FUNCTION_BLOCK CC1SFC
VAR_INPUT
	mode : UINT := 0; //0 = manual, 1=Final conc and total flow set directly
	API_Concentration : LREAL := 1.0; //	API Concentration in mg/mL
	conc : sAnalogConstraint := (sp := 0.0, rq := -100.0, mn := 0.0, mx := 1.0);
	a : sAnalogConstraint := (sp := 0.0, rq := -100.0, mn := 2.0, mx := 70.0);
	b : sAnalogConstraint := (sp := 0.0, rq := -100.0, mn := 20.0, mx := 500.0);
	c : sAnalogConstraint := (sp := 0.0, rq := -100.0, mn := 0.0, mx := 500.0);
END_VAR
VAR_IN_OUT
	FCA : FC1b;
	FTA : AI;
	FCB : FC1b;
	FTB : AI;
	PumpA : sMasterflexPort;
	PumpB : sMasterflexPort;
END_VAR
VAR_OUTPUT
END_VAR
VAR
	cRatio : LREAL;
END_VAR

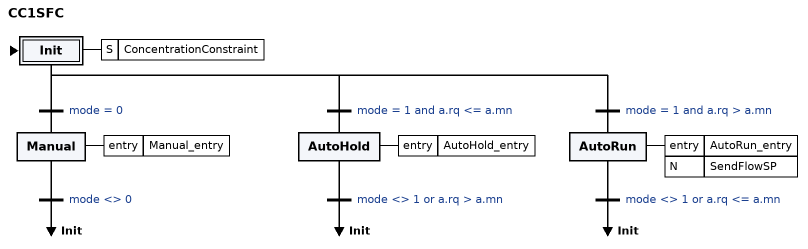
INITIAL_STEP Init:
    ConcentrationConstraint(S);
END_STEP
TRANSITION FROM Init TO Manual
    := mode = 0;
END_TRANSITION
STEP Manual:
    Manual_entry(P1);  // entry action
END_STEP
TRANSITION FROM Manual TO Init
    := mode <> 0;
END_TRANSITION
TRANSITION FROM Init TO AutoHold
    := mode = 1 and a.rq <= a.mn;
END_TRANSITION
STEP AutoHold:
    AutoHold_entry(P1);  // entry action
END_STEP
TRANSITION FROM AutoHold TO Init
    := mode <> 1 or a.rq > a.mn;
END_TRANSITION
TRANSITION FROM Init TO AutoRun
    := mode = 1 and a.rq > a.mn;
END_TRANSITION
STEP AutoRun:
    AutoRun_entry(P1);  // entry action
    SendFlowSP(N);
END_STEP
TRANSITION FROM AutoRun TO Init
    := mode <> 1 or a.rq <= a.mn;
END_TRANSITION

ACTION AutoRun_entry:
//Flow control to Auto
FCA.modeSP := 2; //Auto
FCB.modeSP := 2; //Auto

//Start Pumps
PumpA.nRun_RQ := 1;
PumpA.nRun_RQ := 1;
END_ACTION

ACTION SendFlowSP:
//Set flow controller setpoint to calculated setpoints
FCA.SP := a.sp;
FCB.SP := b.sp;
END_ACTION

ACTION ConcentrationConstraint:
c.mx := a.mx + b.mx;
c.mn := a.mn + b.mn;
a.rq := c.rq * conc.rq/MAX(0.0001,API_Concentration);
b.rq := c.rq - a.rq;
IF a.rq < a.mn OR a.rq > a.mx OR b.rq < b.mn OR b.rq > b.mx OR
   c.rq < c.mn OR c.rq > c.mx OR conc.rq < 0.0 OR conc.rq > API_Concentration THEN
	//calculated flows outside ranges, ignore concentration and total flow requests
	a.rq := a.sp;
	b.rq := b.sp;
	c.rq := c.sp;
	conc.rq := conc.sp;
ELSE
	//flows are in range, change the target to match the request
	a.sp := a.rq;
	b.sp := b.rq;
	c.sp := c.rq;
	conc.sp := conc.rq;
END_IF
END_ACTION

ACTION Manual_entry:
//Bumpless Manual transition
//No actions

//Shutdown Manual transition

//Flow control to Manual
FCA.modeSP := 1; //Manual
FCB.modeSP := 1; //Manual

//Stop Pumps
PumpA.nRun_RQ := 0;
PumpA.nRun_RQ := 0;
END_ACTION

ACTION AutoHold_entry:
//Flow control to Manual
FCA.modeSP := 1; //Manual
FCB.modeSP := 1; //Manual

//Stop Pumps
PumpA.nRun_RQ := 0;
PumpA.nRun_RQ := 0;
END_ACTION

END_FUNCTION_BLOCK

(* stored: Version 1.1.0.1, ProductVersion 3.1.0.36
   POU CC1SFC: Id {abaf130b-ccd7-41fc-afbb-2a37af556628}, SpecialFunc None
   Action AutoRun_entry: Id {05355883-4fae-4428-8d71-3ccb94cc120f}
   Action SendFlowSP: Id {15a68aed-c35a-48c0-9fc3-e4bdf09a5baf}
   Action ConcentrationConstraint: Id {478b6c3c-b213-43e4-8f44-8d4c36f0e249}
   Action Manual_entry: Id {74e0f410-3e3a-43e3-b99f-77d976e06da7}
   Action AutoHold_entry: Id {79111a6b-ef27-46bf-bfdf-78d81718b3a1} *)
